// TwinCAT 3 PLC project FirstPLC
// ProgramVersion: 3.1.4024.0
// libraries:
//   Tc2_Standard, * (Beckhoff Automation GmbH)
//   Tc2_System, * (Beckhoff Automation GmbH)
//   Tc3_Module, * (Beckhoff Automation GmbH)
//   TcUnit, * (www.tcunit.org)
// project tree:
//   / PlcTask.TcTTO, PlcTask2.TcTTO (not stored)
//   POUs/ FB_TestSuite1.TcPOU, FB_TestSuite2.TcPOU, MAIN.TcPOU, PRG_TESTS.TcPOU
// real-time tasks:
//   TASK PlcTask: cycle T#10ms, priority 20, ADS port 350
//   TASK PlcTask2: cycle T#10ms, priority 1, ADS port 351

CONFIGURATION FirstPLC
    RESOURCE PLC ON TwinCAT3
        TASK PlcTask(INTERVAL := T#10ms, PRIORITY := 20);
        PROGRAM MAIN WITH PlcTask : MAIN;
    END_RESOURCE
END_CONFIGURATION

// ---- POUs/MAIN.TcPOU
PROGRAM MAIN
VAR
    bTest : BOOL;
END_VAR

END_PROGRAM

// ---- POUs/FB_TestSuite1.TcPOU
FUNCTION_BLOCK FB_TestSuite1 EXTENDS FB_TestSuite
VAR_INPUT
END_VAR
VAR_OUTPUT
END_VAR
VAR
END_VAR

TestCase1A();
TestCase1BCD();
TestCase1F_IgnoreCase();

METHOD TestCase1BCD
VAR_INPUT
END_VAR
TEST('TestCase1B');

AssertTrue(False, 'Condition is not true');

TEST_FINISHED_NAMED('TestCase1B');

IF TEST_ORDERED('TestCase1C') THEN

    AssertTrue(TRUE, 'Condition is not true');

    TEST_FINISHED();
END_IF

TEST('TestCase1D');

AssertTrue(FALSE, 'Condition is not true');
AssertTrue(TRUE, 'Condition is not true');


TEST_FINISHED();


TEST('TestCase1E with a space');

AssertTrue(TRUE, 'Condition is not true');
AssertTrue(TRUE, 'Condition is not true');


TEST_FINISHED();
END_METHOD

METHOD TestCase1F_IgnoreCase : REFERENCE TO FB_Test
VAR_INPUT
END_VAR
VAR_INST
    step : DINT;
END_VAR

IF TesT_ORdEReD('TestCase1F Ignore Case') THEN
    AssertFalse(False, 'Condition is not false');
    // introduce whitespace for test        
            TEsT_FiNiSHED();
END_IF
END_METHOD

METHOD TestCase1A
VAR_INPUT
END_VAR
TEST('TestCase1A');

AssertTrue(2+2=4, 'Condition is not true');

TEST_FINISHED();
END_METHOD

METHOD TestCase1G_Characters : REFERENCE TO FB_Test
VAR_INPUT
END_VAR
VAR_INST
    step : DINT;
END_VAR

IF TEST_ORDERED('TestCase1G 1*/_-1^&"@!()') THEN
    AssertFalse(TRUE, 'Condition is not false');
    TEST_FINISHED();
END_IF
END_METHOD

END_FUNCTION_BLOCK

// ---- POUs/FB_TestSuite2.TcPOU
FUNCTION_BLOCK FB_TestSuite2 EXTENDS FB_TestSuite
VAR_INPUT
END_VAR
VAR_OUTPUT
END_VAR
VAR
END_VAR

TestCase2A();
TestCase2B();

TEST('TestCase2C');

AssertTrue(TRUE, 'Condition is not true');
AssertTrue(FALSE, 'Condition is not true');

TEST_FINISHED();

METHOD TestCase2A
VAR_INPUT
END_VAR
TEST('TestCase2A');

AssertTrue(TRUE, 'Condition is not true');

TEST_FINISHED();
END_METHOD

METHOD TestCase2B
VAR_INPUT
END_VAR
TEST('TestCase2B');

AssertTrue(TRUE, 'Condition is not true');
AssertTrue(TRUE, 'Condition is not true');

TEST_FINISHED();
END_METHOD

END_FUNCTION_BLOCK

// ---- POUs/PRG_TESTS.TcPOU
PROGRAM PRG_TESTS
VAR
    fbTestSuite1Instance1 : FB_TestSuite1;
    fbTestSuite2Instance1 : FB_TestSuite2;
    fbTestSuite2Instance2 : FB_TestSuite2;
END_VAR

TcUnit.RUN();

END_PROGRAM
